SUBAPPLICATION mapping_blink (* Subapplication Type *)
  (* Standard: 61499-2 *)
  (* Version 1.0, 2023-04-04, franz *)
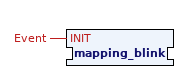
  EVENT_INPUT
    INIT; (* Initialization Request *)
  END_EVENT
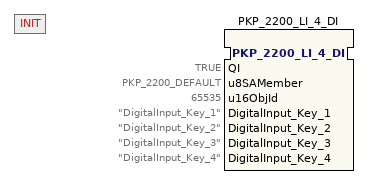
  FBS
    PKP_2200_LI_4_DI : PKP_2200_LI_4_DI(QI := TRUE, u8SAMember := PKP_2200_DEFAULT, u16ObjId := 65535, DigitalInput_Key_1 := "DigitalInput_Key_1", DigitalInput_Key_2 := "DigitalInput_Key_2", DigitalInput_Key_3 := "DigitalInput_Key_3", DigitalInput_Key_4 := "DigitalInput_Key_4");
  END_FBS
END_SUBAPPLICATION
